FUNCTION_BLOCK FB_TwoHandStartCM_Tests EXTENDS TcUnit.FB_TestSuite
VAR
    Device : FB_TwoHandStartCM;
    Hal : ST_TwoHandHal;
    Wired : BOOL;
END_VAR

Release_is_required_between_start_edges();

METHOD Release_is_required_between_start_edges
TEST('Release_is_required_between_start_edges');
IF NOT Wired THEN
    Device.Setup(Name := 'Test.TwoHand', HalRef := Hal);
    Hal.FieldbusHealthy := TRUE;
    Wired := TRUE;
END_IF
Hal.LeftPressed := FALSE; Hal.RightPressed := FALSE; Hal.SafeActive := FALSE;
Device();
AssertTrue(Condition := Device.OutImm.Armed, Message := 'both released arms the functional edge');
Hal.LeftPressed := TRUE; Hal.RightPressed := TRUE; Hal.SafeActive := TRUE;
Device();
AssertTrue(Condition := Device.OutImm.StartPulse, Message := 'certified result rising creates one functional pulse');
Device();
AssertFalse(Condition := Device.OutImm.StartPulse, Message := 'held buttons do not repeat the pulse');
Hal.LeftPressed := FALSE; Hal.RightPressed := FALSE; Hal.SafeActive := FALSE;
Device();
AssertTrue(Condition := Device.OutImm.Armed, Message := 'release rearms the next cycle');
TEST_FINISHED();
END_METHOD

END_FUNCTION_BLOCK

(* stored: Version 1.1.0.1, ProductVersion 3.1.4024.12
   POU FB_TwoHandStartCM_Tests: Id {b2645b4c-e8bf-4913-a40d-3808da3e9515}, SpecialFunc None
   Method Release_is_required_between_start_edges: Id {57c8f489-8eb5-4349-af08-ef08c178a3d6} *)
